PROGRAM JAM_FAULTS
VAR
	TON_GL1_JAM: TON; // MOTOR FAULT DELAY TIMER
	TON_GL2_JAM: TON; // MOTOR FAULT DELAY TIMER
	TON_GL3_JAM: TON; // MOTOR FAULT DELAY TIMER
	TON_GL4_JAM: TON; // MOTOR FAULT DELAY TIMER
	TON_GL5A_JAM: TON; // MOTOR FAULT DELAY TIMER
	TON_GL5B_JAM: TON; // MOTOR FAULT DELAY TIMER
	TON_GL6_JAM: TON; // MOTOR FAULT DELAY TIMER
	TON_GL7_JAM: TON; // MOTOR FAULT DELAY TIMER
	TON_GL8_JAM: TON; // MOTOR FAULT DELAY TIMER
	TON_GL9_JAM: TON; // MOTOR FAULT DELAY TIMER
	TON_GL10_JAM: TON; // MOTOR FAULT DELAY TIMER
	TON_GL11_JAM: TON; // MOTOR FAULT DELAY TIMER
	FAULT_PRESET_TIME: time;
	
			
	GL1: sTransfer;
	GL2: sTransfer;
	GL3: sConveyor;
	GL4: sConveyor;
	GL5: sConveyor;
	GL6: sConveyor;
	GL7:sConveyor;
	GL8: sConveyor;
	GL9: sConveyor;
	GL10: sConveyor;
	GL11: sTransfer;
	GL1_RD: SRoll_Door;
		
END_VAR
VAR // added by the converter: edge detectors and wires of the graphical bodies
    _w1 : BOOL;
END_VAR

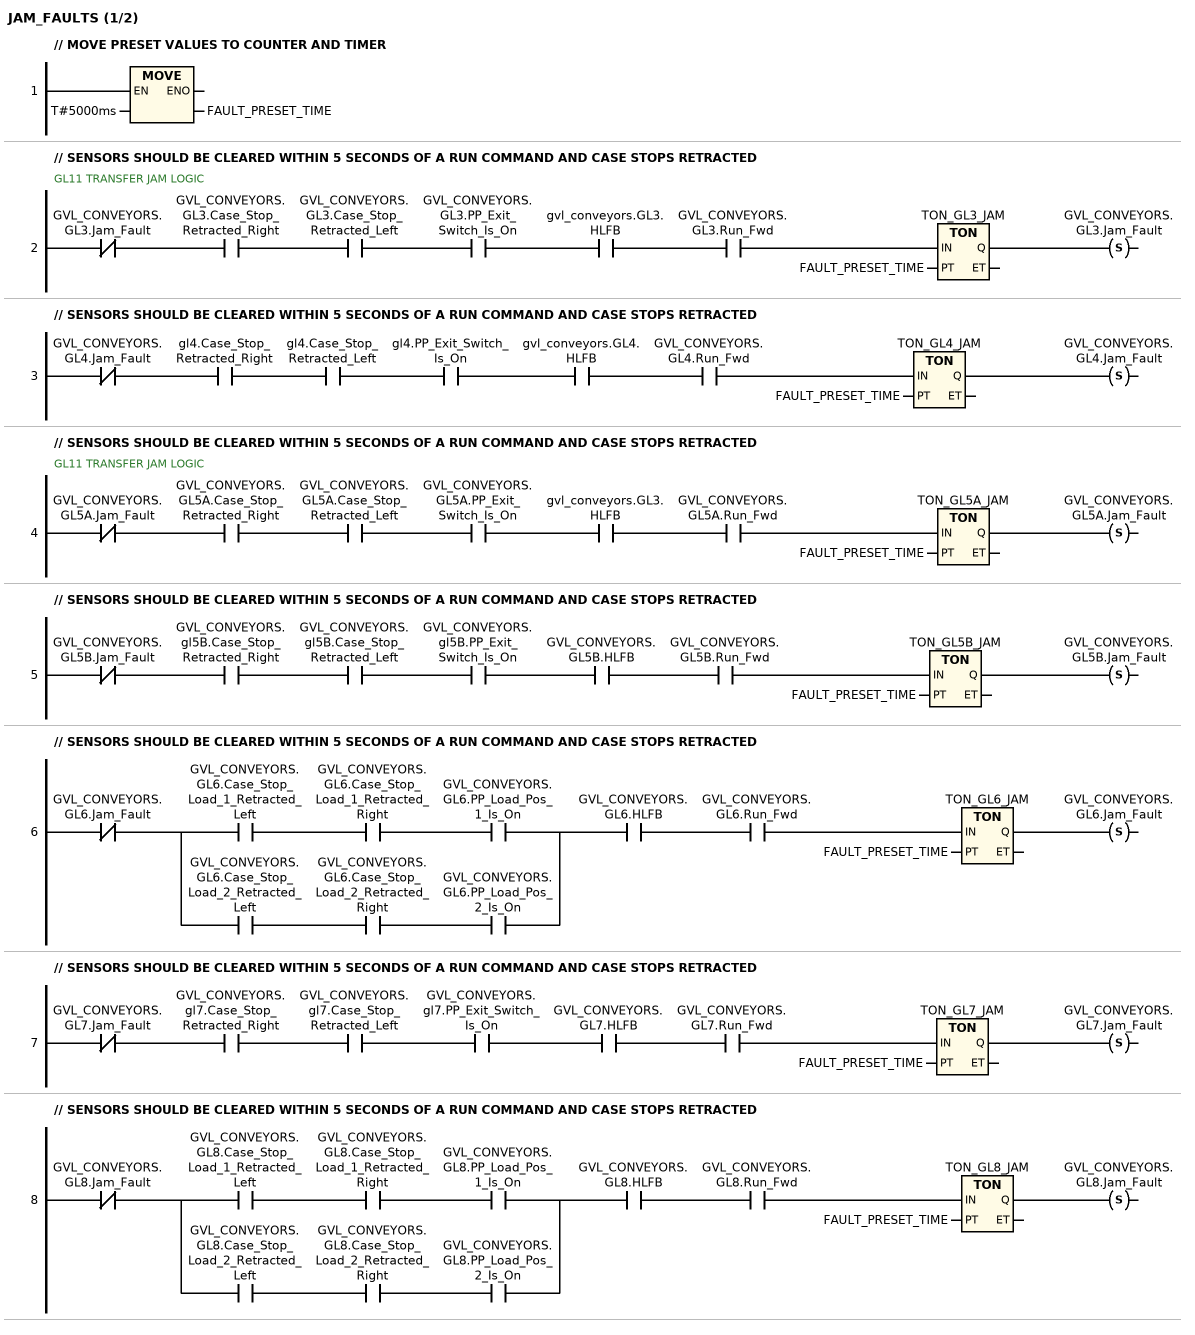
// NETWORK 1: // MOVE PRESET VALUES TO COUNTER AND TIMER
FAULT_PRESET_TIME := T#5000ms;

// NETWORK 2: // SENSORS SHOULD BE CLEARED WITHIN 5 SECONDS OF A RUN COMMAND AND CASE STOPS RETRACTED
// GL11 TRANSFER JAM LOGIC
TON_GL3_JAM(IN := NOT GVL_CONVEYORS.GL3.Jam_Fault AND GVL_CONVEYORS.GL3.Case_Stop_Retracted_Right AND GVL_CONVEYORS.GL3.Case_Stop_Retracted_Left AND GVL_CONVEYORS.GL3.PP_Exit_Switch_Is_On AND gvl_conveyors.GL3.HLFB AND GVL_CONVEYORS.GL3.Run_Fwd, PT := FAULT_PRESET_TIME); // TON
GVL_CONVEYORS.GL3.Jam_Fault S= TON_GL3_JAM.Q;

// NETWORK 3: // SENSORS SHOULD BE CLEARED WITHIN 5 SECONDS OF A RUN COMMAND AND CASE STOPS RETRACTED
TON_GL4_JAM(IN := NOT GVL_CONVEYORS.GL4.Jam_Fault AND gl4.Case_Stop_Retracted_Right AND gl4.Case_Stop_Retracted_Left AND gl4.PP_Exit_Switch_Is_On AND gvl_conveyors.GL4.HLFB AND GVL_CONVEYORS.GL4.Run_Fwd, PT := FAULT_PRESET_TIME); // TON
GVL_CONVEYORS.GL4.Jam_Fault S= TON_GL4_JAM.Q;

// NETWORK 4: // SENSORS SHOULD BE CLEARED WITHIN 5 SECONDS OF A RUN COMMAND AND CASE STOPS RETRACTED
// GL11 TRANSFER JAM LOGIC
TON_GL5A_JAM(IN := NOT GVL_CONVEYORS.GL5A.Jam_Fault AND GVL_CONVEYORS.GL5A.Case_Stop_Retracted_Right AND GVL_CONVEYORS.GL5A.Case_Stop_Retracted_Left AND GVL_CONVEYORS.GL5A.PP_Exit_Switch_Is_On AND gvl_conveyors.GL3.HLFB AND GVL_CONVEYORS.GL5A.Run_Fwd, PT := FAULT_PRESET_TIME); // TON
GVL_CONVEYORS.GL5A.Jam_Fault S= TON_GL5A_JAM.Q;

// NETWORK 5: // SENSORS SHOULD BE CLEARED WITHIN 5 SECONDS OF A RUN COMMAND AND CASE STOPS RETRACTED
TON_GL5B_JAM(IN := NOT GVL_CONVEYORS.GL5B.Jam_Fault AND GVL_CONVEYORS.gl5B.Case_Stop_Retracted_Right AND GVL_CONVEYORS.gl5B.Case_Stop_Retracted_Left AND GVL_CONVEYORS.gl5B.PP_Exit_Switch_Is_On AND GVL_CONVEYORS.GL5B.HLFB AND GVL_CONVEYORS.GL5B.Run_Fwd, PT := FAULT_PRESET_TIME); // TON
GVL_CONVEYORS.GL5B.Jam_Fault S= TON_GL5B_JAM.Q;

// NETWORK 6: // SENSORS SHOULD BE CLEARED WITHIN 5 SECONDS OF A RUN COMMAND AND CASE STOPS RETRACTED
TON_GL6_JAM(IN := NOT GVL_CONVEYORS.GL6.Jam_Fault AND (GVL_CONVEYORS.GL6.Case_Stop_Load_1_Retracted_Left AND GVL_CONVEYORS.GL6.Case_Stop_Load_1_Retracted_Right AND GVL_CONVEYORS.GL6.PP_Load_Pos_1_Is_On OR GVL_CONVEYORS.GL6.Case_Stop_Load_2_Retracted_Left AND GVL_CONVEYORS.GL6.Case_Stop_Load_2_Retracted_Right AND GVL_CONVEYORS.GL6.PP_Load_Pos_2_Is_On) AND GVL_CONVEYORS.GL6.HLFB AND GVL_CONVEYORS.GL6.Run_Fwd, PT := FAULT_PRESET_TIME); // TON
GVL_CONVEYORS.GL6.Jam_Fault S= TON_GL6_JAM.Q;

// NETWORK 7: // SENSORS SHOULD BE CLEARED WITHIN 5 SECONDS OF A RUN COMMAND AND CASE STOPS RETRACTED
TON_GL7_JAM(IN := NOT GVL_CONVEYORS.GL7.Jam_Fault AND GVL_CONVEYORS.gl7.Case_Stop_Retracted_Right AND GVL_CONVEYORS.gl7.Case_Stop_Retracted_Left AND GVL_CONVEYORS.gl7.PP_Exit_Switch_Is_On AND GVL_CONVEYORS.GL7.HLFB AND GVL_CONVEYORS.GL7.Run_Fwd, PT := FAULT_PRESET_TIME); // TON
GVL_CONVEYORS.GL7.Jam_Fault S= TON_GL7_JAM.Q;

// NETWORK 8: // SENSORS SHOULD BE CLEARED WITHIN 5 SECONDS OF A RUN COMMAND AND CASE STOPS RETRACTED
TON_GL8_JAM(IN := NOT GVL_CONVEYORS.GL8.Jam_Fault AND (GVL_CONVEYORS.GL8.Case_Stop_Load_1_Retracted_Left AND GVL_CONVEYORS.GL8.Case_Stop_Load_1_Retracted_Right AND GVL_CONVEYORS.GL8.PP_Load_Pos_1_Is_On OR GVL_CONVEYORS.GL8.Case_Stop_Load_2_Retracted_Left AND GVL_CONVEYORS.GL8.Case_Stop_Load_2_Retracted_Right AND GVL_CONVEYORS.GL8.PP_Load_Pos_2_Is_On) AND GVL_CONVEYORS.GL8.HLFB AND GVL_CONVEYORS.GL8.Run_Fwd, PT := FAULT_PRESET_TIME); // TON
GVL_CONVEYORS.GL8.Jam_Fault S= TON_GL8_JAM.Q;

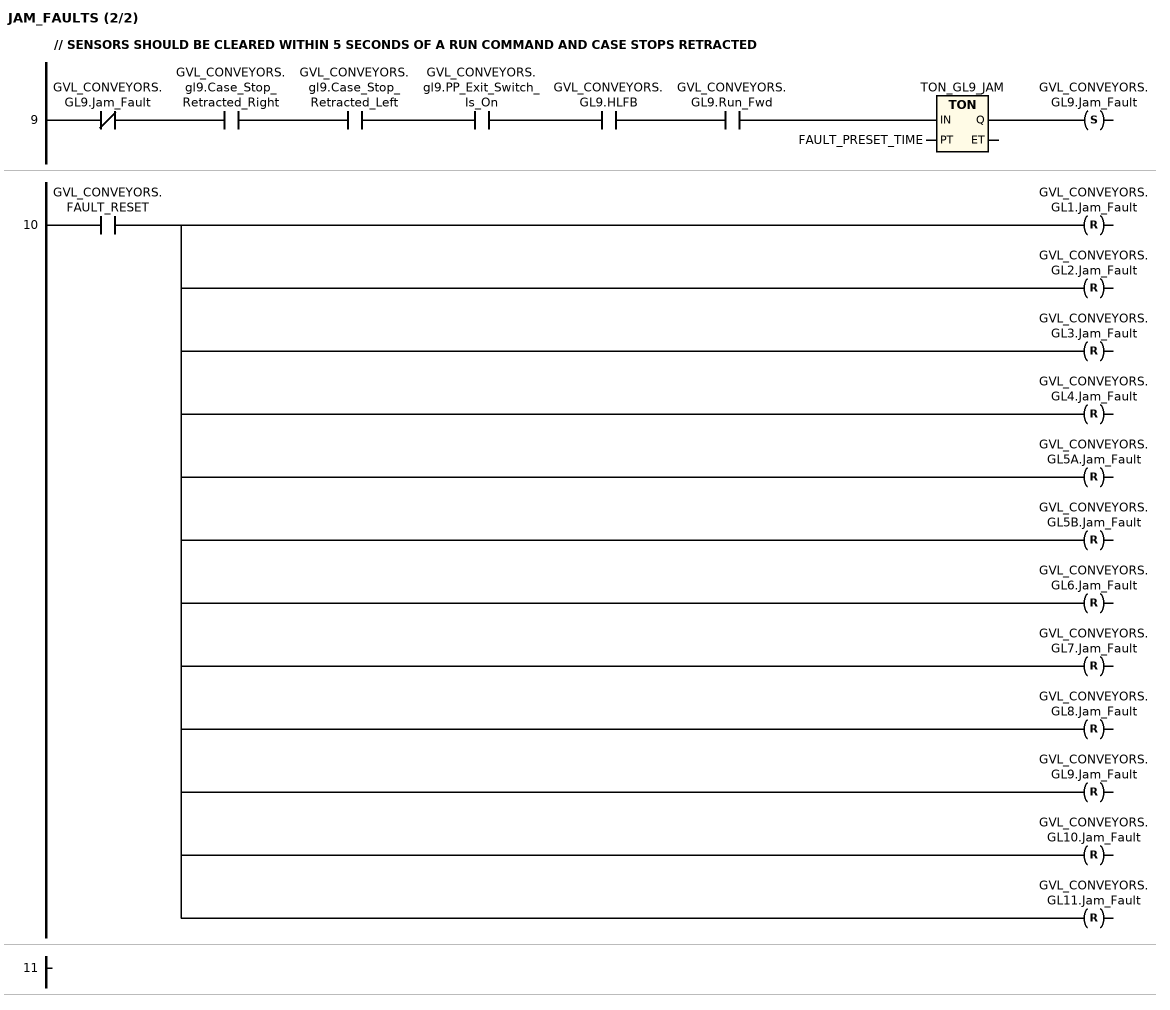
// NETWORK 9: // SENSORS SHOULD BE CLEARED WITHIN 5 SECONDS OF A RUN COMMAND AND CASE STOPS RETRACTED
TON_GL9_JAM(IN := NOT GVL_CONVEYORS.GL9.Jam_Fault AND GVL_CONVEYORS.gl9.Case_Stop_Retracted_Right AND GVL_CONVEYORS.gl9.Case_Stop_Retracted_Left AND GVL_CONVEYORS.gl9.PP_Exit_Switch_Is_On AND GVL_CONVEYORS.GL9.HLFB AND GVL_CONVEYORS.GL9.Run_Fwd, PT := FAULT_PRESET_TIME); // TON
GVL_CONVEYORS.GL9.Jam_Fault S= TON_GL9_JAM.Q;

// NETWORK 10
_w1 := GVL_CONVEYORS.FAULT_RESET;
GVL_CONVEYORS.GL1.Jam_Fault R= _w1;
GVL_CONVEYORS.GL2.Jam_Fault R= _w1;
GVL_CONVEYORS.GL3.Jam_Fault R= _w1;
GVL_CONVEYORS.GL4.Jam_Fault R= _w1;
GVL_CONVEYORS.GL5A.Jam_Fault R= _w1;
GVL_CONVEYORS.GL5B.Jam_Fault R= _w1;
GVL_CONVEYORS.GL6.Jam_Fault R= _w1;
GVL_CONVEYORS.GL7.Jam_Fault R= _w1;
GVL_CONVEYORS.GL8.Jam_Fault R= _w1;
GVL_CONVEYORS.GL9.Jam_Fault R= _w1;
GVL_CONVEYORS.GL10.Jam_Fault R= _w1;
GVL_CONVEYORS.GL11.Jam_Fault R= _w1;

// NETWORK 11

END_PROGRAM

(* stored: Version 1.1.0.1, ProductVersion 3.1.4024.12
   POU JAM_FAULTS: Id {186cd33b-bf35-4a1b-93cc-34a05055d164}, SpecialFunc None *)
